PROGRAM MAIN_FAST
VAR
	i : USINT; (* counter variable *)
END_VAR

(* --------------------------------------------- *)
(* Triamec Motion AG, 6340 Baar, Switzerland     *)
(* Sample Code may be adapted to customer need   *)
(* --------------------------------------------- *)

(* Tria-Link cyclic fast call *)
MAIN.Trialink.CallFast();

(* CNC axis cyclic fast call *)
FOR i := 1 TO MAIN.cAxes DO
	MAIN.Axes[i].Fast();
END_FOR

END_PROGRAM

(* stored: Version 1.1.0.1, ProductVersion 3.1.4024.12
   POU MAIN_FAST: Id {cd456aac-2003-41eb-8d0e-049749eaffb5}, SpecialFunc None *)
